FUNCTION_BLOCK F_TRIG
VAR_INPUT
END_VAR
VAR_OUTPUT
END_VAR
VAR
END_VAR

END_FUNCTION_BLOCK

(* stored: Version 1.1.0.1
   POU F_TRIG: Id {b2a133b3-1cb4-475b-a907-c1dcbe5b4c27}, SpecialFunc None *)
